Staubli VAL3: page_axis.pjx

--- page_axis.pjx ---
Parameters version=s7.2.1 stackSize=5000 millimeterUnit=true
Program file=alreadyExist.pgx
Program file=buildList.pgx
Program file=listAdd.pgx
Program file=loadPage.pgx
Program file=main.pgx
Program file=onBackSpace.pgx
Program file=onDefault.pgx
Program file=onEnterEvent.pgx
Program file=onExit.pgx
Program file=onF1Event.pgx
Program file=onF2Event.pgx
Program file=onF3Event.pgx
Program file=onF4Event.pgx
Program file=onF5Event.pgx
Program file=onF6Event.pgx
Program file=onF7Event.pgx
Program file=onF8Event.pgx
Program file=onStart.pgx
Program file=refresh.pgx
Program file=refreshDynamic.pgx
Program file=refreshStatic.pgx
Program file=showExist.pgx
Data file=page_axis.dtx
Library alias=page path=Disk://kernel/template/page/page.pjx
Library alias=use path=Disk://kernel/userPage/userPage.pjx
Library alias=language path=Disk://kernel/language/language.pjx
Library alias=axis path=Disk://instrSequential/AXIS7/AXIS7.pjx
Library alias=axis8 path=Disk://instrSequential/AXIS8/AXIS8.pjx
Library alias=axis8Move path=Disk://instrSequential/AXIS8/page_axis/page_axis.pjx

--- page_axis.dtx ---
num nTime = 1
num nKey
num nRefresh
num nView
num nIndex
num nPreset[4]
num nSelected
public string sItems
string sMessage
string sMenu[8]
string sList[7]
string sEvent
string sMenu8[8]
bool bButton[8]
bool bLarge
public bool bResetAxis
public aio MbAI_a8Axispose = {link=ModbusSrv-0\Modbus-Word\MbAI_a8Axispose}
public aio MbAI_aCurPosH = {link=ModbusSrv-0\Modbus-Word\MbAI_aCurPosH}
public aio MbAI_aCurPosL = {link=ModbusSrv-0\Modbus-Word\MbAI_aCurPosL}
public aio MbAI_aUnused4 = {link=ModbusSrv-0\Modbus-Word\MbAI_aUnused4}
public aio MbAI_b8MotorErr = {link=ModbusSrv-0\Modbus-Word\MbAI_b8MotorError}
public aio MbAI_b8MotorPow = {link=ModbusSrv-0\Modbus-Word\MbAI_b8MotorPower}
public aio MbAI_bAxis7Reac = {link=ModbusSrv-0\Modbus-Word\MbAI_bAxis7Reached}
public aio MbAI_bAxis8Reac = {link=ModbusSrv-0\Modbus-Word\MbAI_bAxis8Reached}
public aio MbAI_bBackHome = {link=ModbusSrv-0\Modbus-Word\MbAI_bBackHome}
public aio MbAI_bDownLimit = {link=ModbusSrv-0\Modbus-Word\MbAI_bDownLimit}
public aio MbAI_bEndCycl = {link=ModbusSrv-0\Modbus-Word\MbAI_bEndCycl}
public aio MbAI_bHomeDone = {link=ModbusSrv-0\Modbus-Word\MbAI_bHomeDone}
public aio MbAI_bHomeLimit = {link=ModbusSrv-0\Modbus-Word\MbAI_bHomeLimit}
public aio MbAI_bIsHome = {link=ModbusSrv-0\Modbus-Word\MbAI_bIsHome}
public aio MbAI_bMotorErro = {link=ModbusSrv-0\Modbus-Word\MbAI_bMotorError}
public aio MbAI_bMotorPowe = {link=ModbusSrv-0\Modbus-Word\MbAI_bMotorPower}
public aio MbAI_bOutAlarm = {link=ModbusSrv-0\Modbus-Word\MbAI_bOutAlarm}
public aio MbAI_bPowerOn = {link=ModbusSrv-0\Modbus-Word\MbAI_bPowerOn}
public aio MbAI_bStartCycl = {link=ModbusSrv-0\Modbus-Word\MbAI_bStartCycl}
public aio MbAI_bUnused1 = {link=ModbusSrv-0\Modbus-Word\MbAI_bUnused1}
public aio MbAI_bUnused2 = {link=ModbusSrv-0\Modbus-Word\MbAI_bUnused2}
public aio MbAI_bUnused3 = {link=ModbusSrv-0\Modbus-Word\MbAI_bUnused3}
public aio MbAI_bUnused5 = {link=ModbusSrv-0\Modbus-Word\MbAI_bUnused5}
public aio MbAI_bUnused6 = {link=ModbusSrv-0\Modbus-Word\MbAI_bUnused6}
public aio MbAI_bUnused7 = {link=ModbusSrv-0\Modbus-Word\MbAI_bUnused7}
public aio MbAI_bUnused8 = {link=ModbusSrv-0\Modbus-Word\MbAI_bUnused8}
public aio MbAI_bUnused9 = {link=ModbusSrv-0\Modbus-Word\MbAI_bUnused9}
public aio MbAI_bUnused10 = {link=ModbusSrv-0\Modbus-Word\MbAI_bUnused10}
public aio MbAI_bUnused11 = {link=ModbusSrv-0\Modbus-Word\MbAI_bUnused11}
public aio MbAI_bUpLimit = {link=ModbusSrv-0\Modbus-Word\MbAI_bUpLimit}
public aio MbAO_aAxis7Puls = {link=ModbusSrv-0\Modbus-Word\MbAO_aAxis7Pulse}
public aio MbAO_aAxis8Puls = {link=ModbusSrv-0\Modbus-Word\MbAO_aAxis8Pulse}
public aio MbAO_aJogVelo = {link=ModbusSrv-0\Modbus-Word\MbAO_aJogVelo}
public aio MbAO_aJogVelo8 = {link=ModbusSrv-0\Modbus-Word\MbAO_aJogVelo8}
public aio MbAO_aMoveDis = {link=ModbusSrv-0\Modbus-Word\MbAO_aMoveDis}
public aio MbAO_aMoveDis8 = {link=ModbusSrv-0\Modbus-Word\MbAO_aMoveDis8}
public aio MbAO_aMovePosH = {link=ModbusSrv-0\Modbus-Word\MbAO_aMovePosH}
public aio MbAO_aMovePosH8 = {link=ModbusSrv-0\Modbus-Word\MbAO_aMovePosH8}
public aio MbAO_aMovePosL = {link=ModbusSrv-0\Modbus-Word\MbAO_aMovePosL}
public aio MbAO_aMovePosL8 = {link=ModbusSrv-0\Modbus-Word\MbAO_aMovePosL8}
public aio MbAO_aUnused6 = {link=ModbusSrv-0\Modbus-Word\MbAO_aUnused6}
public aio MbAO_aUnused7 = {link=ModbusSrv-0\Modbus-Word\MbAO_aUnused7}
public aio MbAO_aUnused8 = {link=ModbusSrv-0\Modbus-Word\MbAO_aUnused8}
public aio MbAO_aUnused9 = {link=ModbusSrv-0\Modbus-Word\MbAO_aUnused9}
public aio MbAO_aUnused10 = {link=ModbusSrv-0\Modbus-Word\MbAO_aUnused10}
public aio MbAO_aUnused11 = {link=ModbusSrv-0\Modbus-Word\MbAO_aUnused11}
public aio MbAO_aVelocity = {link=ModbusSrv-0\Modbus-Word\MbAO_aVelocity}
public aio MbAO_aVelocity8 = {link=ModbusSrv-0\Modbus-Word\MbAO_aVelocity8}
public aio MbAO_b7Axis = {link=ModbusSrv-0\Modbus-Word\MbAO_b7Axis}
public aio MbAO_b8Axis = {link=ModbusSrv-0\Modbus-Word\MbAO_b8Axis}
public aio MbAO_bAxis7Dire = {link=ModbusSrv-0\Modbus-Word\MbAO_bAxis7Direction}
public aio MbAO_bAxis7Home = {link=ModbusSrv-0\Modbus-Word\MbAO_bAxis7Home}
public aio MbAO_bAxis8Dire = {link=ModbusSrv-0\Modbus-Word\MbAO_bAxis8Direction}
public aio MbAO_bMoveDir = {link=ModbusSrv-0\Modbus-Word\MbAO_bMoveDir}
public aio MbAO_bMoveDirM = {link=ModbusSrv-0\Modbus-Word\MbAO_bMoveDirM}
public aio MbAO_bMovePos8 = {link=ModbusSrv-0\Modbus-Word\MbAO_bMovePos8}
public aio MbAO_bMoveToPos = {link=ModbusSrv-0\Modbus-Word\MbAO_bMoveToPos}
public aio MbAO_bRecordPos = {link=ModbusSrv-0\Modbus-Word\MbAO_bRecordPos}
public aio MbAO_bResetErr = {link=ModbusSrv-0\Modbus-Word\MbAO_bResetErr}
public aio MbAO_bStopMotor = {link=ModbusSrv-0\Modbus-Word\MbAO_bStopMotor}
public aio MbAO_bUnused1 = {link=ModbusSrv-0\Modbus-Word\MbAO_bUnused1}
public aio MbAO_bUnused2 = {link=ModbusSrv-0\Modbus-Word\MbAO_bUnused2}
public aio MbAO_bUnused3 = {link=ModbusSrv-0\Modbus-Word\MbAO_bUnused3}
public aio MbAO_bUnused4 = {link=ModbusSrv-0\Modbus-Word\MbAO_bUnused4}
public aio MbAO_bUnused5 = {link=ModbusSrv-0\Modbus-Word\MbAO_bUnused5}

--- main.pgx ---
public program main()
  local bool l_bSave
begin
  // INIT
  call onStart()
  // LOOP UNTIL nKey=255
  do
    call refresh()
    nKey=getKey()
    call use:listevent(nKey,nIndex,sEvent)
    nView=use:nView
    nSelected=nIndex
    if isKeyPressed(271)
      call onF1Event()
    else
      aioSet(MbAO_bMoveDirM,0)
      aioSet(MbAO_b7Axis,0)
      //logMsg("2")
    endIf
    if isKeyPressed(278)
      call onF8Event()
    else
      aioSet(MbAO_bMoveDir,0)
      aioSet(MbAO_b7Axis,0)
      //logMsg("3")
    endIf

    switch nKey
      case 263
        // backSpace
        call onBackSpace(l_bSave)
      break
      case 259
        // TAB
        bLarge=!bLarge
        call use:setView(bLarge)
      break
     // case 271
     //   call onF1Event()
     // break
      case 272
          call onF2Event()
      break
      case 273
          call onF3Event()
      break
      case 274
        call onF4Event()
      break
      case 275,32
        call onF5Event(l_bSave)
      break
      case 276
        call onF6Event(l_bSave)
      break
      case 277
        call onF7Event(l_bSave)
      break
    //  case 278
     //   call onF8Event(l_bSave)
    //  break
      case 270
        call onEnterEvent(l_bSave)
      break

      default
        call onDefault()
      break
    endSwitch
    // release the resource
    delay(0)
  until nKey==255
  // on Exit
  call onExit(l_bSave)
end

--- alreadyExist.pgx ---
program alreadyExist(string& x_sName[], bool& x_bUndo[])
  local num l_nX
  local num l_nY
  local string l_sString
begin
  l_nX=40-use:nBottomX
  l_nY=use:nBottomY+1
  call language:message(l_sString,21)
  call use:type(l_nX,l_nY,l_sString)
  call use:read(l_nX+len(l_sString),l_nY,x_sName,10,false)
  if !use:bUseEscape
    call axis:find(x_sName,x_bUndo)
    if x_bUndo
      call language:message(x_sName,-2)
      popUpMsg(x_sName)
    endIf
  else
    x_bUndo=true
  endIf
end

--- buildList.pgx ---
program buildList()
  local num l_nSize
  local string l_sEvent
  local num i
  local string l_sString
begin
  // INIT the list
  l_sString=""
  call use:stringCopy(l_sString,sList)
  // Build the list
  call axis:getSize(l_nSize)
  // check the list empty
  call axis:get(l_sEvent,0)
  if l_sEvent!=""
    for i=0 to (l_nSize-1)
      call axis:get(l_sEvent,i)
      if l_sEvent!=""
        call listAdd(toString("2",i+1)+" "+l_sEvent)
      endIf
    endFor
  endIf

end

--- listAdd.pgx ---
program listAdd(string x_sEvent)
begin
  // add in the queue
  if sList!=""
    $dins(sList,size(sList))
  endIf
  sList[size(sList)-1]=x_sEvent
end

--- onBackSpace.pgx ---
program onBackSpace(bool& x_bSave[])
  local string l_sName
  local num l_nX
  local num l_nY
  local string l_sNewName
  local string l_sMessage
  local bool l_bFound
begin
  //
  // NB sEvent is the selected
  // element in the LIST
  //
  // enter the name of the preset
  //
  //if global:mode>0
    call axis:get(l_sName,nIndex)
    // change the name
    if l_sName!=""
      l_nX=40-use:nBottomX+find(sEvent,l_sName)-1
      l_nY=nView+1
      // read the new name string
      l_sNewName=l_sName
      call use:read(l_nX,l_nY,l_sNewName,10,false)
      if l_sName!=l_sNewName and l_sNewName!=""
        call axis:find(l_sNewName,l_bFound)
        if l_bFound
          call language:message(l_sMessage,-2)
        else
          call axis:set(l_sNewName,nIndex)
          x_bSave=true
          call buildList()
        endIf
      endIf
    endIf
  //endIf
end

--- onF1Event.pgx ---
program onF1Event()
  local num l_nJogVelocity
  local num l_nSpeedScale
begin
  // look if the bButton is enable
  if bButton[0]
    // decrease the move


    ////    io:direction_neg=true
    ////    wait(getKey()==-1)
    ////    io:direction_neg=false


//    if ! isPowered()
//       call use:timerDialog("请给手臂上电",1)
//      return
//    endIf

    if aioGet(MbAI_bMotorPowe)==1
      ////7轴负向移动速度
      l_nJogVelocity=100
      ////
      aioSet(MbAO_aJogVelo,l_nJogVelocity)
      aioSet(MbAO_bMoveDirM,1)
      aioSet(MbAO_b7Axis,1)
      call use:timerDialog("7轴负向移动...",0)
    else
      if aioGet(MbAI_bMotorPowe)==0
        call use:timerDialog("7轴未上电",1)
        return
      endIf
    endIf


  endIf
  //

end

--- onF2Event.pgx ---
program onF2Event()
  local num l_nSave
  local string l_sMessage
  local bool l_bYes
  local string l_sButton[2]
begin
  // look if the bButton is enable
  if bButton[1]
    // save the current position

    ////    io:record=true
    ////    delay(0.5)
    ////    io:record=false
    ////    call axis:setValue(aioGet(io:currentPulse),nIndex)

    if aioGet(MbAI_bMotorPowe)==1 and aioGet(MbAI_bBackHome)==1
      l_sMessage="是否要记录当前位置"
      call language:getYesNo(l_sButton)
      call use:yes_no(l_sMessage,l_sButton,l_bYes)
      if l_bYes
        aioSet(MbAO_b7Axis,1)
        aioSet(MbAO_bRecordPos,1)
        delay(0.5)
        aioSet(MbAO_bRecordPos,0)
        aioSet(MbAO_b7Axis,0)
        call axis:setValue(aioGet(MbAI_aCurPosL),nIndex,aioGet(MbAI_aCurPosH))
        l_nSave=axis:libSave()
        if l_nSave==0
          call use:timerDialog("当前位置记录成功",1)
        else
          call use:timerDialog("当前位置记录不成功",1)
        endIf
      endIf
    else
      if aioGet(MbAI_bBackHome)==0
        call use:timerDialog("7轴未回零位",1)
        return
      endIf
      if aioGet(MbAI_bMotorPowe)==0
        call use:timerDialog("7轴未上电",1)
        return
      endIf
    endIf
    //
  endIf
end

--- onF3Event.pgx ---
program onF3Event()
begin
  // look if the bButton is enable
  if bButton[2]
//////////////    // make the calibration
//////////////
//////////////
//////////////    ////    io:calibrate=true
//////////////    ////    delay(0.5)
//////////////    ////    io:calibrate=false
//////////////
//////////////
//////////////    //
//////////////    aioSet(MbAO_b7Axis,1)
//////////////    aioSet(MbAO_bResetErr,1)
//////////////
//////////////    delay(0.5)
//////////////    aioSet(MbAO_b7Axis,0)
//////////////     call use:timerDialog("7轴已经复位",1)
//////////////     bResetAxis=true
//////////////    logMsg("[VALlaser] INTERFACE:7Axis Reset")
     call axis8Move:onF2Event()

  endIf
//  call Axis8Move:onF2Event()
end

--- onF4Event.pgx ---
program onF4Event()
begin
  // look if the bButton is enable
  if bButton[3]
    // go to home


    ////    io:home=true
    ////    delay(0.5)
    ////    io:home=false

    if aioGet(MbAI_bMotorPowe)==1

      call use:timerDialog("Back To Home...",1)
      aioSet(MbAO_bAxis7Home,1)
      aioSet(MbAO_b7Axis,1)
      delay(0.5)
      wait(aioGet(MbAI_bHomeDone)==0 or isKeyPressed(255))
      if isKeyPressed(255)
        aioSet(MbAO_bStopMotor,1)
        delay(0.5)
        aioSet(MbAO_bStopMotor,0)
      endIf
      aioSet(MbAO_b7Axis,0)
    else
      if aioGet(MbAI_bMotorPowe)==0
        call use:timerDialog("7轴未上电",1)
      endIf

    endIf

    //
  endIf
end

--- onF5Event.pgx ---
program onF5Event(bool& x_bSave[])
  local string l_sName
  local string l_sMessage
  local bool l_bYes
  local string l_sButton[2]
begin

  // look if the bButton is enable

  if bButton[4]

    //

    // the simulation is disable when the cycle is active

//    if ! isPowered()

//      call use:timerDialog("请给手臂上电",1)

//      return

//    endIf



    //if !cycleStatus:bCycle

////12.13//////////////      l_sMessage="是否要移动到所选位置"
//////////////////
//////////////////      call language:getYesNo(l_sButton)
//////////////////
//////////////////      call use:yes_no(l_sMessage,l_sButton,l_bYes)
//////////////////
/////12.13/////////////      if l_bYes


///////////////////////////////////bingo!/////////////////////
        call axis:get(l_sName,nIndex)
//          l_sName="PStart"
///////////////////////////////////bingo!/////////////////////
        logMsg("[KERNEL] INTERFACE:Simulation of the: "+"AXIS "+l_sName)

        call use:timerDialog("AXIS  MOVING...",0)

        call axis:onRun(l_sName)


        call use:nullKey(nKey)

        //

        use:bUseRefresh=true

//////12.13//////////      endIf



    //endIf

  endIf

end

--- onF6Event.pgx ---
program onF6Event(bool& x_bSave[])
  local string l_sName
  local num l_nResult
  local string l_sSwap
  local string l_sMessage
  local bool l_bYes
  local string l_sButton[2]
begin
  // look if the bButton is enable
  if bButton[5]
    //
    // delete the selected ITEM
    //
    call axis:get(l_sName,nIndex)
    if l_sName=="workPos"
      call use:timerDialog("该点为系统所有，无法删除",1)
      return
    endIf

    //if nIndex>=0 and global:mode>0
    if nIndex>=0
      call axis:get(l_sName,nIndex)
      if l_sName!=""
        l_sSwap=l_sName="AXIS7>"+l_sName
//        call prog:findItem(l_sSwap,l_nResult,true)
        if l_nResult==0
//          call trajectory:findInstruction(l_sSwap,l_nResult)
          if l_nResult==0
            //delete it
            call language:message(l_sMessage,80)
            call language:getYesNo(l_sButton)
            call use:yes_no(l_sMessage,l_sButton,l_bYes)
            if l_bYes
              call axis:del(nIndex)
              logMsg("[KERNEL] INTERFACE:Delete the AXIS7: "+sEvent+" at position: "+toString("",nIndex))
              // for the refresh
              if nIndex>0
                nIndex=nIndex-1
                if nIndex<nView
                  nView=nIndex
                endIf
              endIf
              nSelected=nIndex
              call buildList()
              call refreshStatic()
              // save it
              x_bSave=true
            endIf
          endIf
        endIf
        if l_nResult!=0
          // TODO
          call showExist(l_sName,l_sSwap)
        endIf
      endIf
    endIf
  endIf

end

--- onF7Event.pgx ---
program onF7Event(bool& x_bSave[])
  local string l_sNew
  local bool l_bUndo
begin
   // look if the bButton is enable
  if bButton[6]
    //
    //  insert a new entry, it's use a FIFO politic
    //
    call alreadyExist(l_sNew,l_bUndo)
    if !l_bUndo and l_sNew!=""
      call axis:new(l_sNew,nIndex+1)
      nSelected=nIndex+1
      call buildList()
      call refreshStatic()
      // save it
      x_bSave=true
    endIf
  endIf
end

--- onF8Event.pgx ---
program onF8Event()
  local num l_nSpeedScale
  local num l_nJogVelocity
begin
  // look if the bButton is enable
  if bButton[7]
    // increase the move

    ////    io:direction_pos=true
    ////    wait(getKey()==-1)
    ////    io:direction_pos=false

//    if ! isPowered()
//       call use:timerDialog("请给手臂上电",1)
//      return
//    endIf
//

    if aioGet(MbAI_bMotorPowe)==1
      //7轴正向移动速度
      l_nJogVelocity=100
      ////
      aioSet(MbAO_aJogVelo,l_nJogVelocity)
      aioSet(MbAO_bMoveDir,1)
      aioSet(MbAO_b7Axis,1)
      call use:timerDialog("7轴正向移动...",0)
    else

      if aioGet(MbAI_bMotorPowe)==0
         call use:timerDialog("7轴未上电",1)
        return
      endIf
    endIf

    //
  endIf
end

--- refreshStatic.pgx ---
program refreshStatic()
  local string l_sMenu
  local string l_sMessage
  local string l_sMotorStatus
begin
  cls()
  //
  // set the view of the page..
  //
  // SET THE PAGE NUMBER
  use:nPage=110
  // load the menu page

  l_sMessage=" -,记录,复位,回零,运动,删除,新建, +"
  //l_sMessage="记录, +, -,校准,回零,运动,删除,新建"

  // define the menu
  call use:stringToArray(l_sMessage,sMenu)
  call use:setMenu(sMenu,true,3)
  call use:getMenu(sMenu,bButton)
  //
  // CREATE THE LIST
  //
  // define your list size for default
  call use:setSizeList(21,0,17,10)
  // set small nParView
  call use:setView(false)
  //
  //call use:listcreate("AXIS7 "+global:sPresetUsing)
  call use:listcreate("AXIS7 ")
  //
  call use:listadd(sList)
  //
  // refresh the cursor
  // select the last item
  call use:selectNewField(nSelected,nIndex,nView)
  if aioGet(MbAI_bBackHome)==1
    l_sMotorStatus="回零位 /"
  else
    l_sMotorStatus="未回零位 /"
  endIf

  if aioGet(MbAI_bMotorErro)==1
    l_sMotorStatus=l_sMotorStatus+" 马达错误"
  else
    l_sMotorStatus=l_sMotorStatus+" 马达正常"
  endIf

  call use:type(0,1,l_sMotorStatus)

end

--- showExist.pgx ---
program showExist(string x_sName, string x_sMessage)
  local string l_sMessage
  local string l_sMessage2
begin
  // not possibile to delete rename
  call language:message(l_sMessage,23)
  call language:message(l_sMessage2,29)
  l_sMessage=l_sMessage+x_sName
  popUpMsg(l_sMessage+l_sMessage2+x_sMessage)
end
